SUBAPPLICATION Uebung_128b_AX (* Übung zu ISOBUS Send Message GLOBAL TP BAM *)
  (* Standard: 61499-2; Description: Copyright (c) 2023 Meisterschulen am Ostbahnhof This program and the accompanying materials are made available under the terms of the Eclipse Public License 2.0 which is available at https://www.eclipse.org/legal/epl-2.0/ SPDX-License-Identifier: EPL-2.0 *)
  (* Version 1.0, 2023-10-23, Franz Höpfinger, Meisterschulen am Ostbahnhof, initial API and implementation and/or initial documentation *)
  PACKAGE Uebungen;
  IMPORT Uebungen::const::Uebung_120_129::Filter::ADD_ALL_PASS;
  IMPORT Uebungen::const::Uebung_120_129::Filter::FLT_ALL_PASS;
  IMPORT isobus::pgn::ADDRESS::GLOBAL_A;
  IMPORT isobus::pgn::ISOUSERHOME_e::thisMember;
  IMPORT isobus::pgn::ISO_CAN_NODE::NODE1;
  IMPORT isobus::pgn::const::PgnDef::PGN_PDU1_PropA;
  IMPORT logiBUS::io::DI::logiBUS_DI::Input_I1;
  IMPORT logiBUS::io::DI::logiBUS_DI_Events::BUTTON_SINGLE_CLICK;
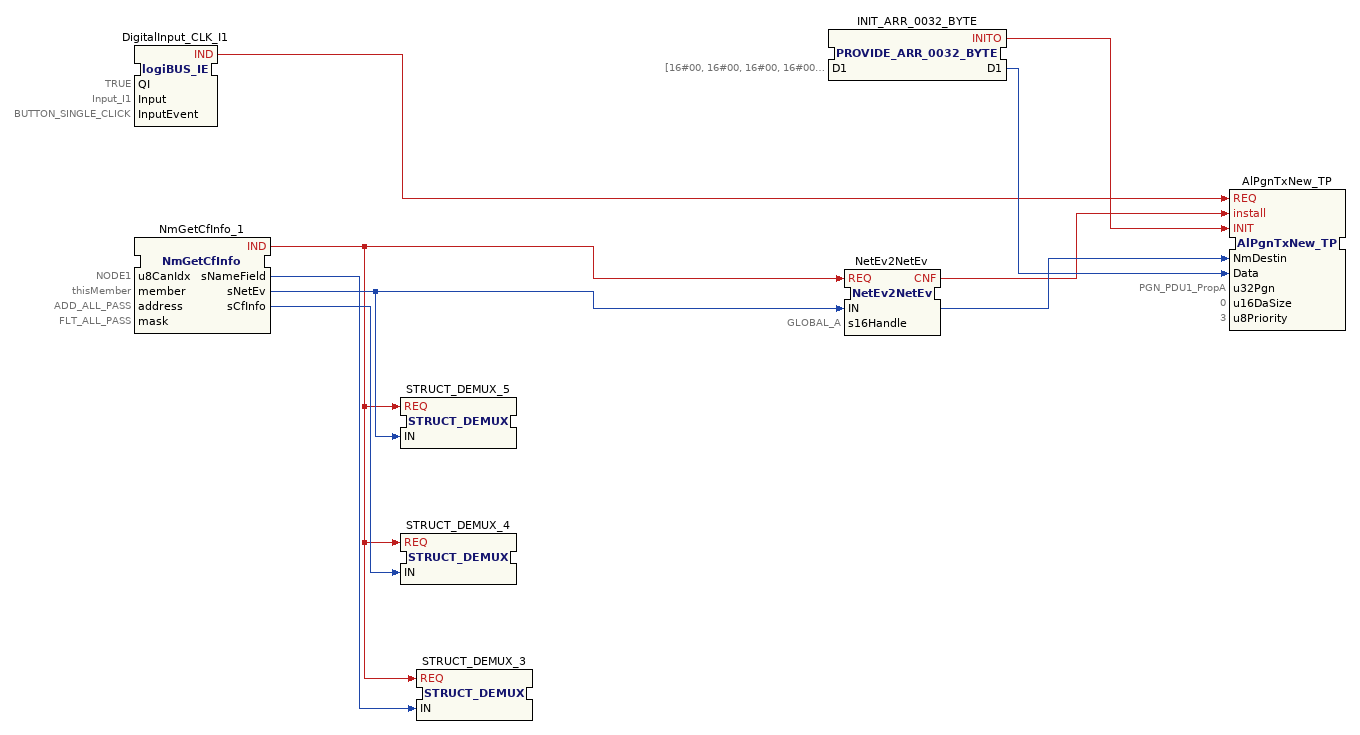
  FBS
    STRUCT_DEMUX_3 : eclipse4diac::convert::STRUCT_DEMUX; {SET_ATTRIBUTE(StructuredType, isobus::pgn::NAMEFIELD_T)}
    NmGetCfInfo_1 : isobus::pgn::NmGetCfInfo(u8CanIdx := NODE1, member := thisMember, address := ADD_ALL_PASS, mask := FLT_ALL_PASS);
    STRUCT_DEMUX_4 : eclipse4diac::convert::STRUCT_DEMUX; {SET_ATTRIBUTE(StructuredType, isobus::pgn::CF_INFO_T)}
    STRUCT_DEMUX_5 : eclipse4diac::convert::STRUCT_DEMUX; {SET_ATTRIBUTE(StructuredType, isobus::pgn::ISONETEVENT_T)}
    AlPgnTxNew_TP : isobus::pgn::tx::AlPgnTxNew_TP(u32Pgn := PGN_PDU1_PropA, u16DaSize := 0, u8Priority := 3);
    DigitalInput_CLK_I1 : logiBUS::io::DI::logiBUS_IE(QI := TRUE, Input := Input_I1, InputEvent := BUTTON_SINGLE_CLICK);
    NetEv2NetEv : isobus::pgn::NetEv2NetEv(s16Handle := GLOBAL_A);
    INIT_ARR_0032_BYTE : eclipse4diac::convert::providers::PROVIDE_ARR_0032_BYTE(D1 := [16#00, 16#00, 16#00, 16#00, 16#00, 16#00, 16#00, 16#00, 16#00, 16#00, 16#00, 16#00, 16#00, 16#00, 16#00, 16#00, 16#00, 16#00, 16#00, 16#00, 16#00, 16#00, 16#00, 16#00, 16#00, 16#00, 16#00, 16#00, 16#00, 16#00, 16#00, 16#00]);
  END_FBS
  EVENT_CONNECTIONS
    NmGetCfInfo_1.IND TO STRUCT_DEMUX_3.REQ;
    NmGetCfInfo_1.IND TO STRUCT_DEMUX_4.REQ;
    NmGetCfInfo_1.IND TO STRUCT_DEMUX_5.REQ;
    NmGetCfInfo_1.IND TO NetEv2NetEv.REQ;
    DigitalInput_CLK_I1.IND TO AlPgnTxNew_TP.REQ;
    NetEv2NetEv.CNF TO AlPgnTxNew_TP.install;
    INIT_ARR_0032_BYTE.INITO TO AlPgnTxNew_TP.INIT;
  END_CONNECTIONS
  DATA_CONNECTIONS
    NmGetCfInfo_1.sNameField TO STRUCT_DEMUX_3.IN;
    NmGetCfInfo_1.sNetEv TO STRUCT_DEMUX_5.IN;
    NmGetCfInfo_1.sCfInfo TO STRUCT_DEMUX_4.IN;
    NmGetCfInfo_1.sNetEv TO NetEv2NetEv.IN;
    NetEv2NetEv. TO AlPgnTxNew_TP.NmDestin;
    INIT_ARR_0032_BYTE.D1 TO AlPgnTxNew_TP.Data;
  END_CONNECTIONS
END_SUBAPPLICATION
